# EPICS substitutions: apps/caenHvApp/Db/seq/dcOnOff.substitutions
file "db/dcOnOff.db" {
pattern { SEC ONOFF VAL }
        { 1 ON 1 }
        { 2 ON 1 }
        { 3 ON 1 }
        { 4 ON 1 }
        { 5 ON 1 }
        { 6 ON 1 }
        { 1 OFF 0 }
        { 2 OFF 0 }
        { 3 OFF 0 }
        { 4 OFF 0 }
        { 5 OFF 0 }
        { 6 OFF 0 }
}
